PROGRAM S5_01_Motion_3
VAR
	HMI_Motion: FB_HMI_Control;
	Motion: FB_Motion2way;

	tMessageOffset: UINT;
	tNumMessagesPerRow: UINT;
	
	
	MyAdvanceInterlock: BOOL;
	MyReturnInterlock: BOOL;
	
	MyAutoAdvanceCondition: BOOL;
	MyAutoReturnCondition: BOOL;
	testword: WORD;
	myAdvancePrompt: BOOL;
	myReturnPrompt: BOOL;
	advancedSensor: BOOL;
	returnedSensor: BOOL;
	AdvanceCoil: BOOL;
	ReturnCoil: BOOL;
	tWaitMsgXICAdv: BOOL;
	tWaitMsgXICRet: BOOL;
END_VAR

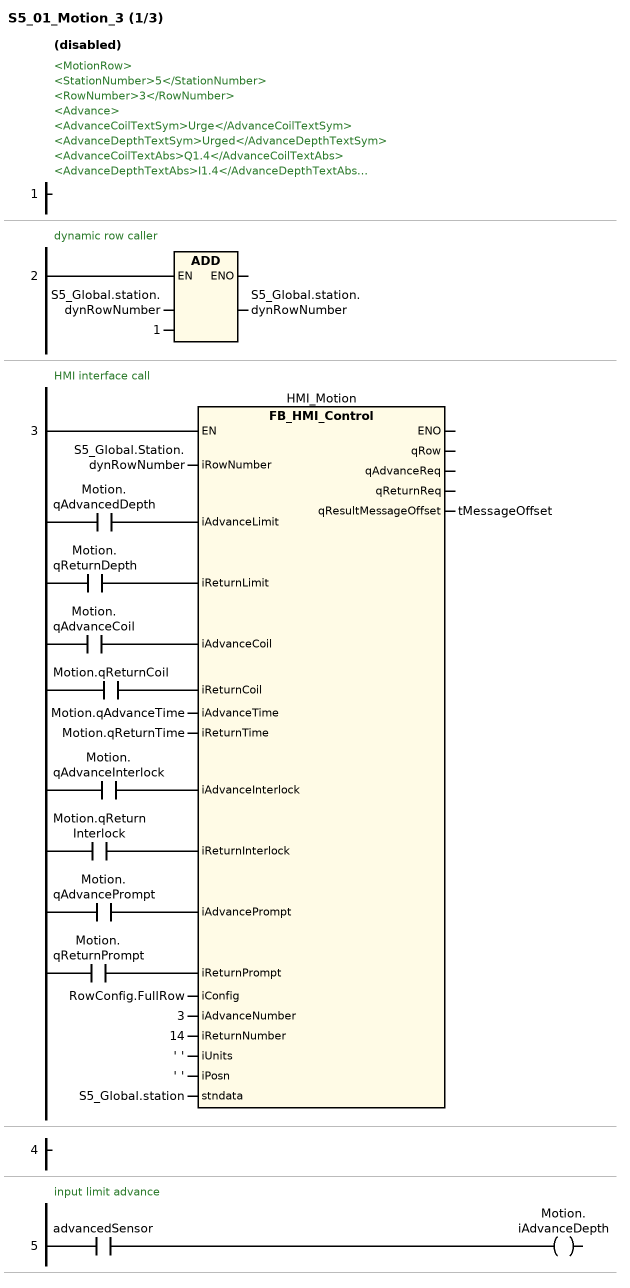
// NETWORK 1 (disabled)
// <MotionRow>
// <StationNumber>5</StationNumber>
// <RowNumber>3</RowNumber>
//   <Advance>
//     <AdvanceCoilTextSym>Urge</AdvanceCoilTextSym>
//     <AdvanceDepthTextSym>Urged</AdvanceDepthTextSym>
//     <AdvanceCoilTextAbs>Q1.4</AdvanceCoilTextAbs>
//     <AdvanceDepthTextAbs>I1.4</AdvanceDepthTextAbs>
//     <ManSeq>5</ManSeq>
//   </Advance>
//   <Return>
//     <ReturnCoilTextSym>Return</ReturnCoilTextSym>
//     <ReturnDepthTextSym>Returned</ReturnDepthTextSym>
//     <ReturnCoilTextAbs>Q1.5</ReturnCoilTextAbs>
//     <ReturnDepthTextAbs>I1.5</ReturnDepthTextAbs>
//    <ManSeq>6</ManSeq>
//   </Return>
//   <Motion>
//     <NameSym>Urger Cylinder</NameSym>
//     <NameAbs>A3</NameAbs>
//   </Motion>
// </MotionRow>

// NETWORK 2
// dynamic row caller
S5_Global.station.dynRowNumber := S5_Global.station.dynRowNumber + 1;

// NETWORK 3
// HMI interface call
HMI_Motion(
    iRowNumber := S5_Global.Station.dynRowNumber,
    iAdvanceLimit := Motion.qAdvancedDepth,
    iReturnLimit := Motion.qReturnDepth,
    iAdvanceCoil := Motion.qAdvanceCoil,
    iReturnCoil := Motion.qReturnCoil,
    iAdvanceTime := Motion.qAdvanceTime,
    iReturnTime := Motion.qReturnTime,
    iAdvanceInterlock := Motion.qAdvanceInterlock,
    iReturnInterlock := Motion.qReturnInterlock,
    iAdvancePrompt := Motion.qAdvancePrompt,
    iReturnPrompt := Motion.qReturnPrompt,
    iConfig := RowConfig.FullRow,
    iAdvanceNumber := 3,
    iReturnNumber := 14,
    iUnits := ' ',
    iPosn := ' ',
    stndata := S5_Global.station,
    qResultMessageOffset => tMessageOffset); // FB_HMI_Control

// NETWORK 4

// NETWORK 5
// input limit advance
Motion.iAdvanceDepth := advancedSensor;

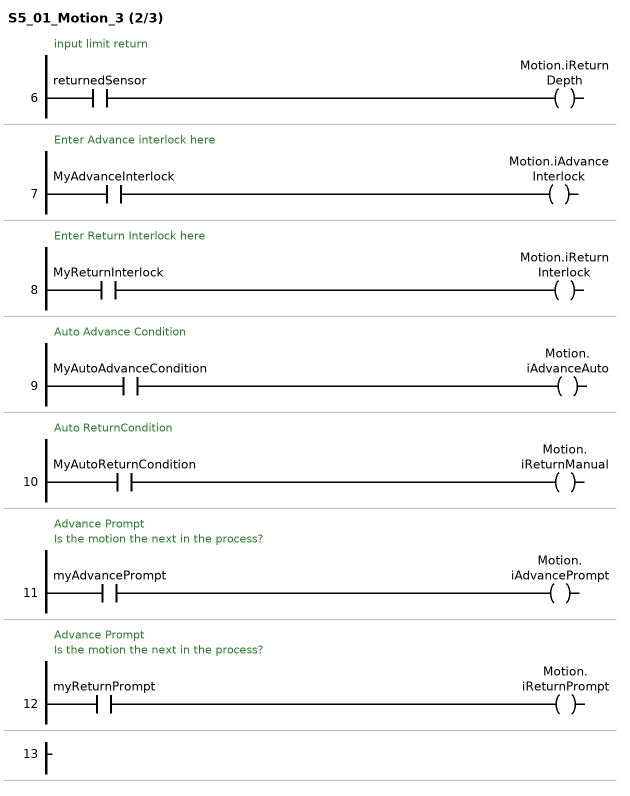
// NETWORK 6
// input limit return
Motion.iReturnDepth := returnedSensor;

// NETWORK 7
// Enter Advance interlock here
Motion.iAdvanceInterlock := MyAdvanceInterlock;

// NETWORK 8
// Enter Return Interlock here
Motion.iReturnInterlock := MyReturnInterlock;

// NETWORK 9
// Auto Advance Condition
Motion.iAdvanceAuto := MyAutoAdvanceCondition;

// NETWORK 10
// Auto ReturnCondition
Motion.iReturnManual := MyAutoReturnCondition;

// NETWORK 11
// Advance Prompt
// Is the motion the next in the process?
Motion.iAdvancePrompt := myAdvancePrompt;

// NETWORK 12
// Advance Prompt
// Is the motion the next in the process?
Motion.iReturnPrompt := myReturnPrompt;

// NETWORK 13

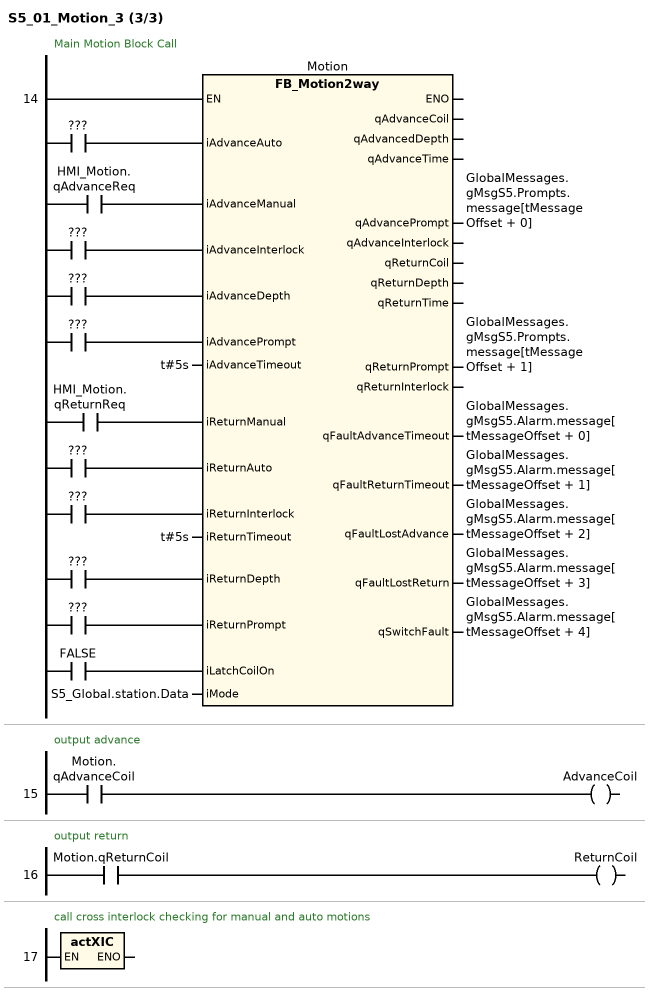
// NETWORK 14
// Main Motion Block Call
Motion(
    iAdvanceManual := HMI_Motion.qAdvanceReq,
    iAdvanceTimeout := t#5s,
    iReturnManual := HMI_Motion.qReturnReq,
    iReturnTimeout := t#5s,
    iLatchCoilOn := FALSE,
    iMode := S5_Global.station.Data,
    qAdvancePrompt => GlobalMessages.gMsgS5.Prompts.message[tMessageOffset + 0],
    qReturnPrompt => GlobalMessages.gMsgS5.Prompts.message[tMessageOffset + 1],
    qFaultAdvanceTimeout => GlobalMessages.gMsgS5.Alarm.message[tMessageOffset + 0],
    qFaultReturnTimeout => GlobalMessages.gMsgS5.Alarm.message[tMessageOffset + 1],
    qFaultLostAdvance => GlobalMessages.gMsgS5.Alarm.message[tMessageOffset + 2],
    qFaultLostReturn => GlobalMessages.gMsgS5.Alarm.message[tMessageOffset + 3],
    qSwitchFault => GlobalMessages.gMsgS5.Alarm.message[tMessageOffset + 4]); // FB_Motion2way

// NETWORK 15
// output advance
AdvanceCoil := Motion.qAdvanceCoil;

// NETWORK 16
// output return
ReturnCoil := Motion.qReturnCoil;

// NETWORK 17
// call cross interlock checking for manual and auto motions
actXIC();

ACTION actXIC:
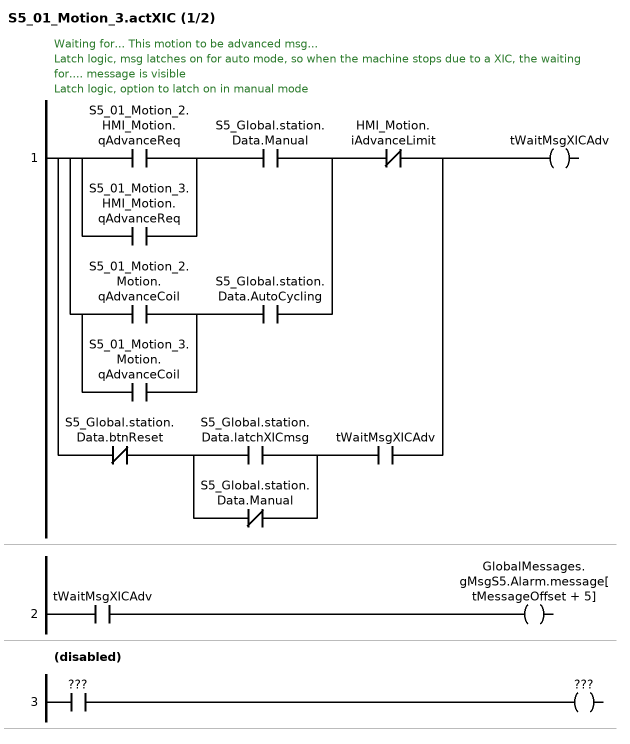
// NETWORK 1
// Waiting for... This motion to be advanced msg...
// Latch logic, msg latches on for auto mode, so when the machine stops due to a XIC, the waiting for.... message is visible
// Latch logic, option to latch on in manual mode
tWaitMsgXICAdv := ((S5_01_Motion_2.HMI_Motion.qAdvanceReq OR S5_01_Motion_3.HMI_Motion.qAdvanceReq) AND S5_Global.station.Data.Manual OR (S5_01_Motion_2.Motion.qAdvanceCoil OR S5_01_Motion_3.Motion.qAdvanceCoil) AND S5_Global.station.Data.AutoCycling) AND NOT HMI_Motion.iAdvanceLimit OR NOT S5_Global.station.Data.btnReset AND (S5_Global.station.Data.latchXICmsg OR NOT S5_Global.station.Data.Manual) AND tWaitMsgXICAdv;

// NETWORK 2
GlobalMessages.gMsgS5.Alarm.message[tMessageOffset + 5] := tWaitMsgXICAdv;

// NETWORK 3 (disabled)
// ??? := ???;

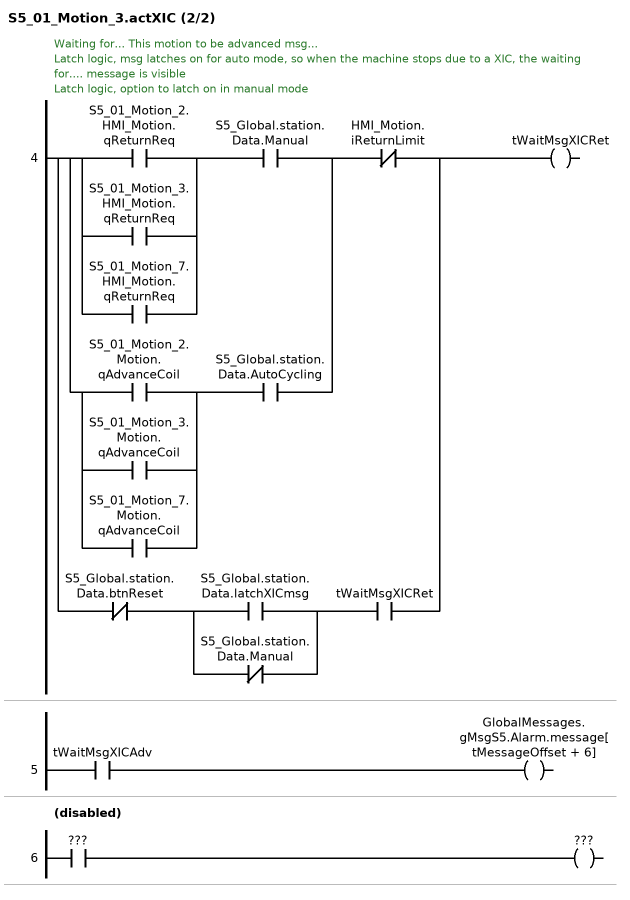
// NETWORK 4
// Waiting for... This motion to be advanced msg...
// Latch logic, msg latches on for auto mode, so when the machine stops due to a XIC, the waiting for.... message is visible
// Latch logic, option to latch on in manual mode
tWaitMsgXICRet := ((S5_01_Motion_2.HMI_Motion.qReturnReq OR S5_01_Motion_3.HMI_Motion.qReturnReq OR S5_01_Motion_7.HMI_Motion.qReturnReq) AND S5_Global.station.Data.Manual OR (S5_01_Motion_2.Motion.qAdvanceCoil OR S5_01_Motion_3.Motion.qAdvanceCoil OR S5_01_Motion_7.Motion.qAdvanceCoil) AND S5_Global.station.Data.AutoCycling) AND NOT HMI_Motion.iReturnLimit OR NOT S5_Global.station.Data.btnReset AND (S5_Global.station.Data.latchXICmsg OR NOT S5_Global.station.Data.Manual) AND tWaitMsgXICRet;

// NETWORK 5
GlobalMessages.gMsgS5.Alarm.message[tMessageOffset + 6] := tWaitMsgXICAdv;

// NETWORK 6 (disabled)
// ??? := ???;
END_ACTION

END_PROGRAM

(* stored: Version 1.1.0.1, ProductVersion 3.1.4024.11
   POU S5_01_Motion_3: Id {739b8195-89b5-09fe-1245-6d4a85e19ca3}, SpecialFunc None
   Action actXIC: Id {ca74de58-1983-018a-2d22-dbb816a93590} *)
